// TIA Portal V20 export
DATA_BLOCK "HmiInterface"   // DB160
// stored: Access Published, MemoryReserve 100, Namespace Unit1.Em2
   VAR
      em : "LAF_typeEmInterface";
      emHomedCheck : "Unit1.Em2.typeEmHomedCheck";
      semiAutoSplice : "LER_typeSequenceInterface";
   END_VAR
   VAR RETAIN
      cmElectrodeFixRightTopFwdBwd : "LBC_typeTwoWayActuatorInterface";
      cmElectrodeFixRightBottomFwdBwd : "LBC_typeTwoWayActuatorInterface";
      cmElectrodeFixLeftTopFwdBwd : "LBC_typeTwoWayActuatorInterface";
      cmElectrodeFixLeftBottomFwdBwd : "LBC_typeTwoWayActuatorInterface";
      cmElectrodeFixLeftTopUpDown : "LBC_typeTwoWayActuatorInterface";
      cmElectrodeFixLeftBottomUpDown : "LBC_typeTwoWayActuatorInterface";
      cmUwSemiSplicerVacuumRightTopOnOff : "LBC_typeTwoWayActuatorInterface";
      cmUwSemiSplicerVacuumRightBottomOnOff : "LBC_typeTwoWayActuatorInterface";
      cmUwSemiSplicerVacuumLeftTopOnOff : "LBC_typeTwoWayActuatorInterface";
      cmUwSemiSplicerVacuumLeftBottomOnOff : "LBC_typeTwoWayActuatorInterface";
      cmElectrodeCutterFwdBwd : "LBC_typeTwoWayActuatorInterface";
      cmSplicingLeftModuleMoverFwdBwd : "LBC_typeTwoWayActuatorInterface";
      cmSplicingRightModuleMoverFwdBwd : "LBC_typeTwoWayActuatorInterface";
      cmElectrodeLeftHolderMoverFwdBwd : "LBC_typeTwoWayActuatorInterface";
      cmElectrodeRightHolderMoverFwdBwd : "LBC_typeTwoWayActuatorInterface";
      cmTapeLoadingTurnCwCcw : "LBC_typeTwoWayActuatorInterface";
      cmTapeAttachUnitFwdBwd : "LBC_typeTwoWayActuatorInterface";
      cmTapeVacuumOnOff : "LBC_typeTwoWayActuatorInterface";
      cmStopperFwdBwd : "LBC_typeTwoWayActuatorInterface";
      cmSupportUnitTransferFwdBwd : "LBC_typeTwoWayActuatorInterface";
      cmSupportUnitShaftUpDown : "LBC_typeTwoWayActuatorInterface";
      cmFrameCoverFwdBwd : "LBC_typeTwoWayActuatorInterface";
   END_VAR
   VAR
      cmUwSemiSplicing1Times : Bool;
   END_VAR
BEGIN
END_DATA_BLOCK
